FUNCTION_BLOCK logiBUS_AI_ID (* Input service interface function block for double word input data *)
  (* Description: Copyright (c) 2017 fortiss GmbH, HR Agrartechnik GmbH This program and the accompanying materials are made available under the terms of the Eclipse Public License 2.0 which is available at https://www.eclipse.org/legal/epl-2.0/ SPDX-License-Identifier: EPL-2.0 AnalogInput_hysteresis = 0 switches the change trigger off (use 1 to see every change). TimeDelta = 0 or 16#FFFFFFFF switches the cyclic IND off. With both off the block sends no IND (value only via REQ). IN = 0-4095 (12 bit, fixed full-scale raw value, ESP32-P4 ADC continuous/DMA mode has no other bit width to choose from). *)
  (* Version 1.1, 2026-04-19, Franz Höpfinger, HR Agrartechnik GmbH *)
  (* Version 1.0, 2017-03-20, Monika Wenger, fortiss GmbH *)
  PACKAGE logiBUS::io::AI;
  (* Documentation:
  logiBUS_AI_ID
   🇩🇪 Deutsch
   Service-Interface-Funktionsblock für die Verarbeitung eines einzelnen analogen Eingangs (Double-Word). Der Baustein bindet einen physischen logiBUS-Analogeingang (Input_I1..I8) ein und liefert dessen Rohwert zyklisch oder änderungsbasiert über IN zurück.
   Schnittstelle
    - INIT (mit QI, PARAMS, Input, AnalogInput_hysteresis, TimeDelta, TimeRateLimit): Initialisiert den Service und wählt den physischen Eingang.
   - REQ (mit QI): Fordert eine sofortige Abfrage des aktuellen Werts an.
   - INITO (mit QO, STATUS): Bestätigt die Initialisierung.
   - CNF (mit QO, STATUS, IN): Antwort auf REQ.
   - IND (mit QO, STATUS, IN): Asynchrone Indikation bei zyklischer oder änderungsbasierter Aktualisierung.
    Roh-Vollausschlag von IN
   IN liefert den Rohwert des ADC als DWORD im Bereich 0-4095 (12 bit). Auf dem ESP32-P4 ist dieser Bereich im verwendeten Continuous/DMA-ADC-Modus fix — es gibt keine andere wählbare Bit-Breite (SOC_ADC_DIGI_MIN_BITWIDTH = SOC_ADC_DIGI_MAX_BITWIDTH = 12).
   Umrechnung Rohwert → Volt: Vout = Dout × Vmax / 4096 (Vmax abhängig von der ADC-Dämpfung ADC_ATTEN_DB_12).
   Hysterese und Zeitsteuerung
   Ein IND wird aus zwei unabhängigen Gründen ausgelöst:
    - Änderung: Weicht der Rohwert um mehr als AnalogInput_hysteresis vom zuletzt gemeldeten Wert ab, kommt ein IND, frühestens TimeRateLimit ms nach dem letzten IND (TimeRateLimit 0 = ohne Begrenzung). AnalogInput_hysteresis = 0 schaltet diesen Auslöser ab; wer jede Änderung sehen will, setzt 1.
   - Zyklisch: Spätestens alle TimeDelta ms kommt ein IND mit dem aktuellen Wert. TimeDelta = 0 oder 16#FFFFFFFF schaltet diesen Auslöser ab.
    Sind beide Auslöser abgeschaltet (AnalogInput_hysteresis = 0 und TimeDelta = 0 bzw. 16#FFFFFFFF), liefert der Baustein keine IND-Ereignisse mehr; der Wert ist dann nur noch über REQ abfragbar. Beim INIT erscheint in diesem Fall eine Warnung im Log.
   🇬🇧 English
   Service interface function block for processing a single analog input (double word). The block wraps a physical logiBUS analog input (Input_I1..I8) and returns its raw value either cyclically or on change via IN.
   Interface
    - INIT (with QI, PARAMS, Input, AnalogInput_hysteresis, TimeDelta, TimeRateLimit): Initializes the service and selects the physical input.
   - REQ (with QI): Requests an immediate read of the current value.
   - INITO (with QO, STATUS): Confirms initialization.
   - CNF (with QO, STATUS, IN): Response to REQ.
   - IND (with QO, STATUS, IN): Asynchronous indication on cyclic or change-based update.
    Raw full-scale value of IN
   IN delivers the raw ADC value as a DWORD in the range 0-4095 (12 bit). On the ESP32-P4, this range is fixed in the continuous/DMA ADC mode used here — no other bit width can be selected (SOC_ADC_DIGI_MIN_BITWIDTH = SOC_ADC_DIGI_MAX_BITWIDTH = 12).
   Raw-to-volt conversion: Vout = Dout × Vmax / 4096 (Vmax depends on the ADC attenuation ADC_ATTEN_DB_12).
   Hysteresis and timing
   An IND is triggered for two independent reasons:
    - Change: When the raw value differs from the last reported value by more than AnalogInput_hysteresis, an IND is sent, at the earliest TimeRateLimit ms after the previous IND (TimeRateLimit 0 = no limit). AnalogInput_hysteresis = 0 switches this trigger off; to see every change, use 1.
   - Cyclic: An IND with the current value is sent at least every TimeDelta ms. TimeDelta = 0 or 16#FFFFFFFF switches this trigger off.
    With both triggers off (AnalogInput_hysteresis = 0 and TimeDelta = 0 or 16#FFFFFFFF) the block sends no IND events at all; the value can then only be read via REQ. A warning is logged at INIT in that case.
  *)
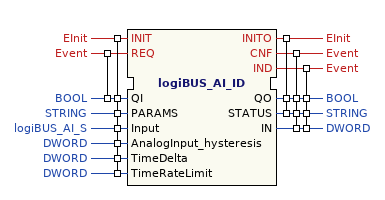
  EVENT_INPUT
    INIT : EInit WITH QI, PARAMS, Input, AnalogInput_hysteresis, TimeDelta, TimeRateLimit; (* Service Initialization *)
    REQ WITH QI; (* Service Request *)
  END_EVENT
  EVENT_OUTPUT
    INITO : EInit WITH QO, STATUS; (* Initialization Confirm *)
    CNF WITH QO, STATUS, IN; (* Confirmation of Requested Service *)
    IND WITH QO, STATUS, IN; (* Indication from Resource *)
  END_EVENT
  VAR_INPUT
    QI : BOOL; (* Event Input Qualifier *)
    PARAMS : STRING; (* Service Parameters *)
    Input : logiBUS::io::AI::logiBUS_AI_S := logiBUS_AI::Invalid; (* Identify the Input Input_I1..I8 *)
    AnalogInput_hysteresis : DWORD; (* IND when the raw value changes by more than this (0 = off) *)
    TimeDelta : DWORD := 250; (* After How many ms an IND (poll interval, 0 or 16#FFFFFFFF = off) *)
    TimeRateLimit : DWORD := 100; (* Maximum 1 IND in how many ms. (< delta) *)
  END_VAR
  VAR_OUTPUT
    QO : BOOL; (* Event Output Qualifier *)
    STATUS : STRING; (* Service Status *)
    IN : DWORD; (* Input data from resource, raw value 0-4095 (12 bit, fixed ESP32-P4 ADC continuous-mode full scale) *)
  END_VAR
END_FUNCTION_BLOCK
